DATA_BLOCK "DT-Chars_DB"
VAR
  Sum_Days : Int;
  Sum_Year : Int;
END_VAR
BEGIN
END_DATA_BLOCK
